// TIA Portal project "drives test" (V17)

(* hardware
DEVICE "S7-1200 station_1"  S7-1200 Station
   slot 0: "Rack_0"  S7-1200 Rack  Rack  V1.0
   slot 1: "PLC_1"  CPU 1214C DC/DC/DC  6ES7 214-1AG40-0XB0  V4.2
DEVICE "HMI_1"  KTP700 Basic PN
   slot 0: "HMI_1"  KTP700 Basic PN  6AV2 123-2GB03-0AX0  15.0.0.0
   slot 1: "HMI_RT_1"  KTP700 Basic PN  6AV2 123-2GB03-0AX0  15.0.0.0
   slot 5: "HMI_1.IE_CP_1"  PROFINET Interface  15.0.0.0
      slot 1: "PROFINET Interface_1"  PROFINET Interface
         slot 1: "Port_1"  Port
DEVICE "SCALANCE X005"  SCALANCE X-Station
   slot 0: "SCALANCE X rack"  Rail
   slot 0: "Switch_1"  6GK5 005-0BA00-1AB2  V1.0
DEVICE "ET 200SP station_1"  ET 200SP-Station
   slot 0: "Rack_0"  Rack  6ES5 710-8MAx1
   slot 0: "IO device_1"  IM 155-6 PN/2 HF  6ES7 155-6AU01-0CN0  V4.2
   slot 1: "DQ 8x24VDC/0.5A HF_1"  DQ 8x24VDC/0.5A HF  6ES7 132-6BF00-0CA0  V2.0
      slot 1: "DQ 8x24VDC/0.5A HF_1"  DQ 8x24VDC/0.5A HF
   slot 2: "DQ 8x24VDC/0.5A HF_2"  DQ 8x24VDC/0.5A HF  6ES7 132-6BF00-0CA0  V2.0
      slot 1: "DQ 8x24VDC/0.5A HF_2"  DQ 8x24VDC/0.5A HF
   slot 3: "DI 8x24VDC HF_1"  DI 8x24VDC HF  6ES7 131-6BF00-0CA0  V2.0
      slot 1: "DI 8x24VDC HF_1"  DI 8x24VDC HF
   slot 4: "DI 8x24VDC HF_2"  DI 8x24VDC HF  6ES7 131-6BF00-0CA0  V2.0
      slot 1: "DI 8x24VDC HF_2"  DI 8x24VDC HF
   slot 5: "DI 8x24VDC HF_3"  DI 8x24VDC HF  6ES7 131-6BF00-0CA0  V2.0
      slot 1: "DI 8x24VDC HF_3"  DI 8x24VDC HF
   slot 6: "Server module_1"  Server module  6ES7 193-6PA00-0AA0  V1.1
      slot 1: "Server module_1"  Server module
   slot 127: "BA 2xRJ45"  BA 2xRJ45  6ES7 193-6AR00-0AA0  V0.0
      slot 1: "Port_1"  X1 P1 R  6ES7 193-6AR00-0AA0  V0.0
      slot 2: "Port_2"  X1 P2 R  6ES7 193-6AR00-0AA0  V0.0
DEVICE "GSD device_1"  GSD.Device.PN
   slot 0: "Rack"  Rack  V1.0
   slot 0: "drivexb14fe3"  SINAMICS G120 CU250S-2 PN Vector V4.7  6SL3 246-0BA22-1FAx  V4.70
      slot 0: "SINAMICS G120 CU250S-2 PN Vector V4.7"  SINAMICS G120 CU250S-2 PN Vector V4.7
      slot 1: "PN-IO"  PN-IO
         slot 1: "Port 1"  Port 1
         slot 2: "Port 2"  Port 2
      slot 1: "DO VECTOR_1"  DO VECTOR
         slot 0: "Module Access Point"  Module Access Point
   slot 2: "Standard telegram 1, PZD-2/2"  Standard telegram 1, PZD-2/2
*)

// ===== PLC "PLC_1"  CPU 1214C DC/DC/DC =====

VAR_GLOBAL   // PLC tag table "Default tag table"
   "Tag_1" AT %QW64 : Word;
   "Tag_2" AT %QW66 : Int;
END_VAR

TYPE "HMI_TAGS"
   STRUCT
      START : Bool;
      STOP : Bool;
      ENABLE : Bool;
      FOWARD : Bool;
      REVERSE : Bool;
      RUN : Bool;
      RUNNING : Bool;
      INC : Bool;
      DEC : Bool;
   END_STRUCT;
END_TYPE

DATA_BLOCK "HMI"   // DB1
{ S7_Optimized_Access := 'TRUE' }
VERSION : 0.1
   VAR
      HMI : "HMI_TAGS";
   END_VAR
BEGIN
END_DATA_BLOCK

// folder: System blocks/Program resources

DATA_BLOCK "IEC_Counter_0_DB"   // DB2
{ S7_Optimized_Access := 'TRUE' }
AUTHOR : Simatic
FAMILY : IEC
NAME : CNTR
VERSION : 1.0
// stored: InstanceOfName IEC_COUNTER
"IEC_COUNTER"
BEGIN
END_DATA_BLOCK

// folder: (top level)

ORGANIZATION_BLOCK "Main"   // OB1, LAD, ProgramCycle
TITLE = "Main Program Sweep (Cycle)"
{ S7_Optimized_Access := 'TRUE' }
VERSION : 0.1
   VAR_INPUT
      Initial_Call : Bool;   // Initial call of this OB
      Remanence : Bool;   // =True, if remanent data are available
   END_VAR
BEGIN

REGION Network 1
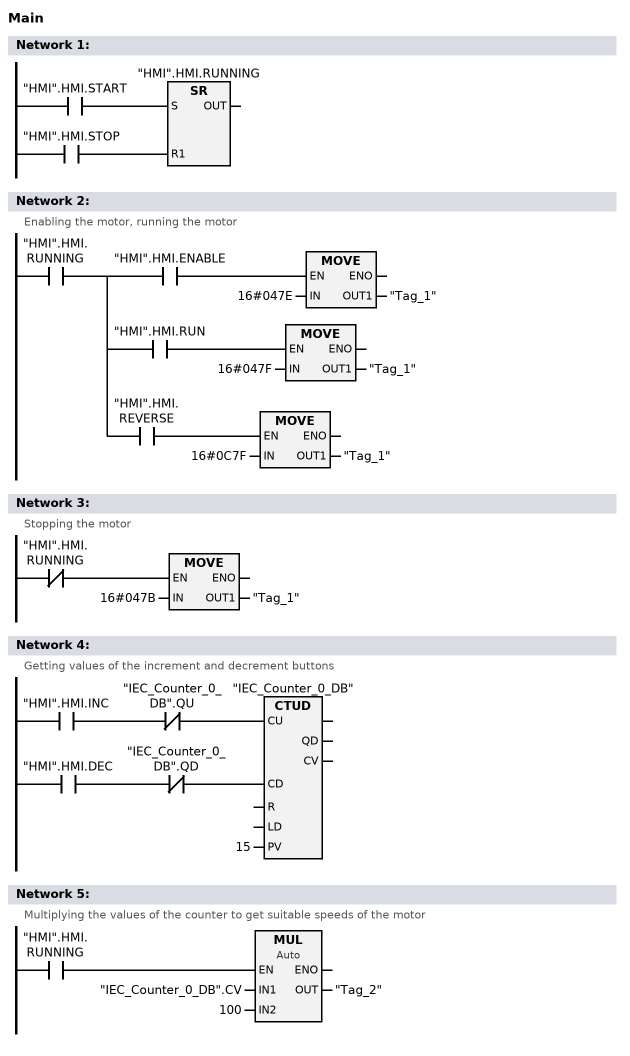
   RUNG wire#powerrail
      Contact( "HMI".HMI.START )
      S_SR(operand := "HMI".HMI.RUNNING, r1 := wire#w1)
   END_RUNG
   RUNG wire#powerrail
      Contact( "HMI".HMI.STOP )
   END_RUNG wire#w1
   // the same network as SCL:
   IF "HMI".HMI.START THEN
       "HMI".HMI.RUNNING := TRUE;   // SR flip-flop
   END_IF;
   IF "HMI".HMI.STOP THEN "HMI".HMI.RUNNING := FALSE; END_IF;
END_REGION

REGION Network 2
   // Enabling the motor, running the motor
   RUNG wire#powerrail
      Contact( "HMI".HMI.RUNNING )
      wire#w1
      Contact( "HMI".HMI.ENABLE )
      Move(in := 16#047E, out1 => "Tag_1")
   END_RUNG
   RUNG wire#w1
      Contact( "HMI".HMI.RUN )
      Move(in := 16#047F, out1 => "Tag_1")
   END_RUNG
   RUNG wire#w1
      Contact( "HMI".HMI.REVERSE )
      Move(in := 16#0C7F, out1 => "Tag_1")
   END_RUNG
   // the same network as SCL:
   IF "HMI".HMI.RUNNING AND "HMI".HMI.ENABLE THEN "Tag_1" := 16#047E; END_IF;
   IF "HMI".HMI.RUNNING AND "HMI".HMI.RUN THEN "Tag_1" := 16#047F; END_IF;
   IF "HMI".HMI.RUNNING AND "HMI".HMI.REVERSE THEN "Tag_1" := 16#0C7F; END_IF;
END_REGION

REGION Network 3
   // Stopping the motor
   RUNG wire#powerrail
      I_Contact( "HMI".HMI.RUNNING )
      Move(in := 16#047B, out1 => "Tag_1")
   END_RUNG
   // the same network as SCL:
   IF NOT "HMI".HMI.RUNNING THEN "Tag_1" := 16#047B; END_IF;
END_REGION

REGION Network 4
   // Getting values of the increment and decrement buttons
   "IEC_Counter_0_DB".CTUD(CU := "HMI".HMI.INC AND NOT "IEC_Counter_0_DB".QU,
                           CD := "HMI".HMI.DEC AND NOT "IEC_Counter_0_DB".QD,
                           PV := 15);
END_REGION

REGION Network 5
   // Multiplying the values of the counter to get suitable speeds of the motor
   RUNG wire#powerrail
      Contact( "HMI".HMI.RUNNING )
      Mul(in1 := "IEC_Counter_0_DB".CV, in2 := 100, out => "Tag_2")
   END_RUNG
   // the same network as SCL:
   IF "HMI".HMI.RUNNING THEN "Tag_2" := "IEC_Counter_0_DB".CV * 100; END_IF;
END_REGION
END_ORGANIZATION_BLOCK

(* ===== HMI "HMI_RT_1" =====
system functions are stored by id; their names below are inferred from use
connection "HMI_Connection_1": ETHERNET, SMART_S7_1200_OMS

HMI tags "Default tag table"
   "HMI_HMI" : HMI_TAGS = PLC HMI.HMI, 1 s

screen "Screen_1" 800x480
   Button "Button_1" at 98,39 size 158x55; TextOff 'START'
      on Press: SetBit("START")
      on Release: ResetBit("START")
   Button "Button_2" at 98,118 size 158x55; TextOff 'STOP'
      on Release: ResetBit("STOP")
      on Press: SetBit("STOP")
   Button "Button_3" at 95,197 size 158x55; TextOff 'ENABLE'
      on Release: ResetBit("ENABLE")
      on Press: SetBit("ENABLE")
   Circle "Circle_1" at 534,184 size 109x109
      Appearance <- "RUNNING"
   Button "Button_4" at 95,293 size 158x55; TextOff 'RUN'
      on Release: ResetBit("RUN")
      on Press: SetBit("RUN")
   Button "Button_5" at 98,373 size 158x55; TextOff 'REVERSE'
      on Release: ResetBit("REVERSE")
      on Press: SetBit("REVERSE")
   Button "Button_6" at 460,73 size 96x32; TextOff '--'
      on Press: SetBit("DEC")
      on Release: ResetBit("DEC")
   Button "Button_7" at 631,74 size 96x32; TextOff '++'
      on Press: SetBit("INC")
      on Release: ResetBit("INC")
*)